FUNCTION_BLOCK GF_Ruehren EXTENDS FB_Basisfunktionalitaeten
VAR_INPUT
	// Instanzieren von Sensoren mit Interfaces
	
	// Instanzieren von Aktoren mit Interfaces
	Ruehrer		:I_Motor1R;
	
	
	// Fragen
	// Wo definiere ich die gewschwindigkeit oder wie kommt diese zum Funktionsblock? 
	// Wird die Geschwindigkeit über den Shrittablauf definiert? 
END_VAR
VAR_OUTPUT
	
END_VAR
VAR
	
END_VAR

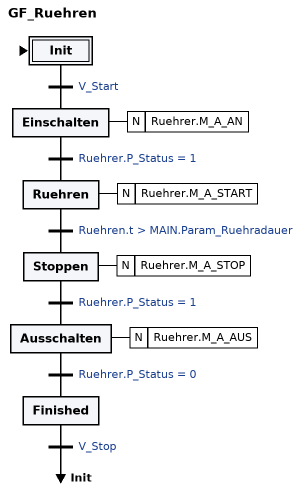
INITIAL_STEP Init:
END_STEP
TRANSITION FROM Init TO Einschalten
    := V_Start;
END_TRANSITION
STEP Einschalten:
    Ruehrer.M_A_AN(N);
END_STEP
TRANSITION FROM Einschalten TO Ruehren
    := Ruehrer.P_Status = 1;
END_TRANSITION
STEP Ruehren:
    Ruehrer.M_A_START(N);
END_STEP
TRANSITION FROM Ruehren TO Stoppen
    := Ruehren.t > MAIN.Param_Ruehradauer;
END_TRANSITION
STEP Stoppen:
    Ruehrer.M_A_STOP(N);
END_STEP
TRANSITION FROM Stoppen TO Ausschalten
    := Ruehrer.P_Status = 1;
END_TRANSITION
STEP Ausschalten:
    Ruehrer.M_A_AUS(N);
END_STEP
TRANSITION FROM Ausschalten TO Finished
    := Ruehrer.P_Status = 0;
END_TRANSITION
STEP Finished:
END_STEP
TRANSITION FROM Finished TO Init
    := V_Stop;
END_TRANSITION

END_FUNCTION_BLOCK

(* stored: Version 1.1.0.1, ProductVersion 3.1.4024.12
   POU GF_Ruehren: Id {715003b6-7dcf-4be3-a0ad-5b1a6bf337c1}, SpecialFunc None *)
